Staubli VAL3: action_wait.pgx

program action_wait()
  local bool l_bEmpty
begin
  // wait no action on the list
  while l_bEmpty==false
    call cycleStatus:isActionEmpty(l_bEmpty)
    delay(0)
  endWhile
end
